# EPICS StreamDevice protocol: streamDevice/leds.proto
# Sidekick EPICS LEDs protocol file
# Built by examining examples at: https://paulscherrerinstitute.github.io/StreamDevice/protocol.html#gen

Terminator = CR LF;

info {
	ExtraInput = Ignore;
	out "*IDN?";
	in "%39c";
}

# Brightness is an integer, 0 to 255
# Use long integer record type
getBrightness {
        out "BRIGhtness:LED\$1?";
        in "%i";
    }

setBrightness {
        out "BRIGhtness:LED\$1 %i";
        @init { getBrightness; }
    }

# Duration is an unsigned long integer
# Use int64 record type
getDuration {
        out "DURation:LED\$1?";
        in "%i";
    }

setDuration {
        out "DURation:LED\$1 %i";
        @init { getDuration; }
    }

debug {
   ExtraInput = Ignore;
   out "%s";
   in "%39c";
}
